FUNCTION_BLOCK T_ExampleMOduleProductionMode EXTENDS T_BaseMode IMPLEMENTS I_PackMode
VAR_INPUT
END_VAR
VAR_OUTPUT
END_VAR
VAR
//  ComponentsCollection : I_ComponentsCollection;
//  xAxis : I_ComponentBase;
  //_modeInterface : I_PackML_BaseModule;
  _specificEquipmentIWantToUse : I_ExampleEquipment;
END_VAR

{warning 'add method implementation '}
METHOD Aborted
END_METHOD

{warning 'add method implementation '}
METHOD Aborting
END_METHOD

{warning 'add method implementation '}
METHOD Clearing
END_METHOD

{warning 'add method implementation '}
METHOD Complete
END_METHOD

{warning 'add method implementation '}
METHOD Completing
END_METHOD

{warning 'add method implementation '}
METHOD Execute
cartesianRobot.PickFromStagingArea();


//THEN OTHER LOGIC
END_METHOD

METHOD GenericInit
VAR_INPUT
  _mode : I_PackML_BaseModule;
END_VAR
// obvs needs more error checking code.

_modeInterface := _mode;
IF NOT __QUERYINTERFACE(_mode, _specificEquipmentIWantToUse) THEN
  ; // ERRROR
END_IF
END_METHOD

{warning 'add method implementation '}
METHOD Held
END_METHOD

{warning 'add method implementation '}
METHOD Holding
END_METHOD

{warning 'add method implementation '}
METHOD Idle
END_METHOD

{warning 'add method implementation '}
METHOD Resetting
END_METHOD

{warning 'add method implementation '}
METHOD Starting
END_METHOD

{warning 'add method implementation '}
METHOD Stopped
END_METHOD

{warning 'add method implementation '}
METHOD Stopping
END_METHOD

{warning 'add method implementation '}
METHOD Suspended
END_METHOD

{warning 'add method implementation '}
METHOD Suspending
END_METHOD

{warning 'add method implementation '}
METHOD Unholding
END_METHOD

{warning 'add method implementation '}
METHOD Unsuspending
END_METHOD

END_FUNCTION_BLOCK

(* stored: Version 1.1.0.1, ProductVersion 3.1.4024.12
   POU T_ExampleMOduleProductionMode: Id {5ca1db18-c049-43e8-9b0c-d88e02f7cfeb}, SpecialFunc None
   Method Aborted: Id {72e04fed-0681-46e7-bca4-6e94e10d452f}
   Method Aborting: Id {7e1f6f19-b21e-4b6b-8be1-2c8a7a49e27d}
   Method Clearing: Id {7d21eb07-7fb9-42b9-8850-69b666656420}
   Method Complete: Id {5f8ee395-dd9a-4ed3-962a-d97836f033a6}
   Method Completing: Id {d1b52729-e6cc-4535-a1f3-38f67eea795e}
   Method Execute: Id {1088d2f4-c779-47d9-a851-81ccc7652da5}
   Method GenericInit: Id {c4e6b5a8-1c9a-401e-9125-cd1690eaa8de}
   Method Held: Id {8fecb6a2-8d5e-4bf3-98f1-12ad08f4f8ae}
   Method Holding: Id {47678e7e-0833-452f-81fc-2d04abe07814}
   Method Idle: Id {3a068a2c-4610-4f61-a951-8ffa4dfcae5b}
   Method Resetting: Id {3db451a8-b105-47e2-9de5-289c94721a88}
   Method Starting: Id {6d7f16f3-12a5-492f-be6b-1f41669a9a20}
   Method Stopped: Id {9ceda6d2-f072-46a2-8651-a643cd7a3cb2}
   Method Stopping: Id {1ce06ec2-2c99-4c87-b978-cad2b5aa1302}
   Method Suspended: Id {e2976bb3-b3b6-4eab-b559-de272a5ecba3}
   Method Suspending: Id {e3592235-f418-4893-8d5c-66481368a04a}
   Method Unholding: Id {8982bdc5-63ba-41c1-ab13-2919737f732f}
   Method Unsuspending: Id {32a72db5-0b20-4d20-8f47-225a7f72a5eb} *)
